ABB RAPID module: MY_Module.sysx

MODULE MY_Module(SYSMODULE)
    TASK PERS num myM_Number := 10;

    PROC myM_Proc()
        TPWrite "My module procedure called...";
    ENDPROC
ENDMODULE
